TYPE T_OHM_Filename : STRING(44);
END_TYPE

(* stored: Version 1.1.0.1
   DUT T_OHM_Filename: Id {eb053653-4fa9-4cf6-a3d9-60e01adc4a2f} *)
